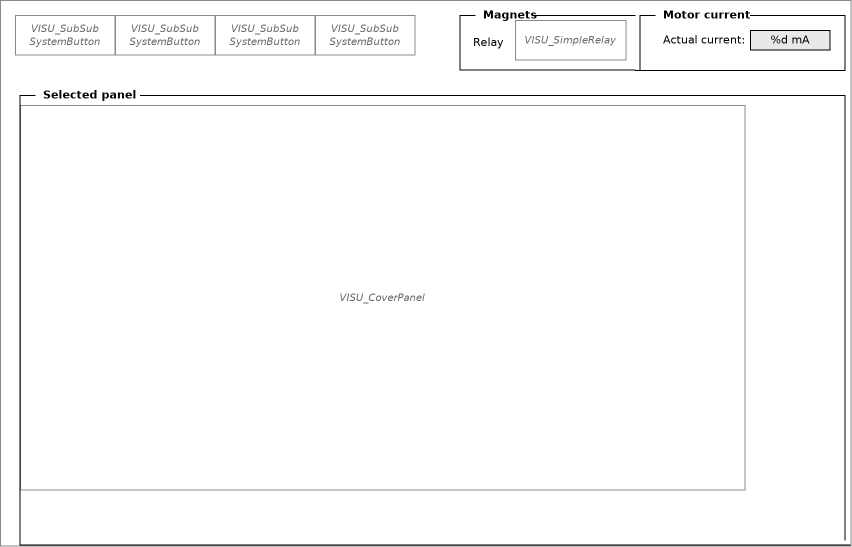
VISUALIZATION VISU_CoverPanelSet  // 852x547
VAR_IN_OUT
	config : CoverPanelSetConfig;
	set : CoverPanelSet;
    widget : CoverPanelSetWidget;
    currentMeasurement : CurrentMeasurement;
END_VAR
    Frame (515,20 111x40)
        shows VISU_SimpleRelay(ref := set.parts.magnetsRelay, widget := widget.magnetsRelay)
    Frame (15,15 100x40)
        shows VISU_SubSubSystemButton(widget := widget.button_p1)
        OnMouseClick: FrameSelectionChange Selection=SelectedFrame=36dcb027-776f-4b31-acd8-d66c3f6e2cf1, GlobSel=AssignType=Directly, SelType=Locally
        OnMouseClick: execute { widget.activeTab := 0; }
    Frame (115,15 100x40)
        shows VISU_SubSubSystemButton(widget := widget.button_p2)
        OnMouseClick: FrameSelectionChange Selection=SelectedFrame=36dcb027-776f-4b31-acd8-d66c3f6e2cf1, Selection=1, GlobSel=AssignType=Directly, SelType=Locally
        OnMouseClick: execute { widget.activeTab := 1; }
    Frame (215,15 100x40)
        shows VISU_SubSubSystemButton(widget := widget.button_p3)
        OnMouseClick: FrameSelectionChange Selection=SelectedFrame=36dcb027-776f-4b31-acd8-d66c3f6e2cf1, Selection=2, GlobSel=AssignType=Directly, SelType=Locally
        OnMouseClick: execute { widget.activeTab := 2; }
    Frame (315,15 100x40)
        shows VISU_SubSubSystemButton(widget := widget.button_p4)
        OnMouseClick: FrameSelectionChange Selection=SelectedFrame=36dcb027-776f-4b31-acd8-d66c3f6e2cf1, Selection=3, GlobSel=AssignType=Directly, SelType=Locally
        OnMouseClick: execute { widget.activeTab := 3; }
    Frame (20,105 725x385), frame switch variable: widget.activeTab
        shows VISU_CoverPanel(panelConfig := config.p1, panel := set.parts.p1, widget := widget.p1)
        shows VISU_CoverPanel(panelConfig := config.p2, panel := set.parts.p2, widget := widget.p2)
        shows VISU_CoverPanel(panelConfig := config.p3, panel := set.parts.p3, widget := widget.p3)
        shows VISU_CoverPanel(panelConfig := config.p4, panel := set.parts.p4, widget := widget.p4)
    Line (20,95) (35,95)
    Label (40,85 100x20), "Selected panel"
    Line (140,95) (845,95)
    Line (845,540) (845,95)
    Line (850,545) (20,545)
    Line (20,545) (20,95)
    Label (470,25 55x35), "Relay"
    Line (460,15) (475,15)
    Label (480,5 100x20), "Magnets"
    Line (535,15) (635,15)
    Line (640,70) (640,15)
    Line (635,70) (460,70)
    Line (460,70) (460,15)
    Label (660,20 90x40), "Actual current:"
    Rectangle (750,30 80x20), "%d mA", text variable: currentMeasurement.current.milliAmps.value, colour toggle: currentMeasurement.statuses.healthStatus.bad
    Line (845,70) (845,15)
    Label (660,5 100x20), "Motor current"
    Line (640,15) (655,15)
    Line (750,15) (845,15)
    Line (635,70) (845,70)
END_VISUALIZATION

(* stored: Version 1.1.0.1, ProductVersion 3.1.4019.2
   Visu VISU_CoverPanelSet: Id {5fa58630-5dcd-42ca-834b-eae69de6e55b} *)
